TYPE ST_PositionParameters : // Full positioning command parameters
STRUCT
	fTargetPos		: LREAL;
	fVelocity		: LREAL;
	fAcceleration	: LREAL;
	fDeceleration	: LREAL; 
	fJerk			: LREAL;
	eBuffermode		: MC_BufferMode;
END_STRUCT
END_TYPE

(* stored: Version 1.1.0.1
   DUT ST_PositionParameters: Id {23ef4253-cd80-4a86-aeab-c62bc6a2bc6e} *)
